TYPE E_EcDiacStatus :
(

	eEcDiac_Start							:= 0, 
	eEcDiac_Delay							,
	eEcDiac_ReadMasterState					,
	eEcDiac_ReadSlaveState

);
END_TYPE
(* End *)

(* stored: Version 1.1.0.1, ProductVersion 3.1.4020.3
   DUT E_EcDiacStatus: Id {d074548a-a206-4230-b593-2f17dc266e17} *)
